// TIA Portal V16 export
// export: Created 2022-01-12T14:34:25.3404927Z, ExportSetting WithDefaults, DisplayName Totally Integrated Automation Portal, DisplayVersion V16 Update 4, DisplayName TIA Portal Version Control Interface, DisplayVersion V16 Update 2, DisplayName TIA Portal Openness, DisplayVersion V16 Update 4, DisplayName STEP 7 Professional, DisplayVersion V16 Update 4, DisplayName STEP 7 Safety, DisplayVersion V16, DisplayName WinCC Professional, DisplayVersion V16 Update 4
VAR_GLOBAL   // PLC tag table "Default tag table"
   System_Byte AT %MB1 : Byte;
   FirstScan AT %M1.0 : Bool;
   DiagStatusUpdate AT %M1.1 : Bool;
   AlwaysTRUE AT %M1.2 : Bool;
   AlwaysFALSE AT %M1.3 : Bool;
   Clock_Byte AT %MB0 : Byte;
   Clock_10Hz AT %M0.0 : Bool;
   Clock_5Hz AT %M0.1 : Bool;
   "Clock_2.5Hz" AT %M0.2 : Bool;
   Clock_2Hz AT %M0.3 : Bool;
   "Clock_1.25Hz" AT %M0.4 : Bool;
   Clock_1Hz AT %M0.5 : Bool;
   "Clock_0.625Hz" AT %M0.6 : Bool;
   "Clock_0.5Hz" AT %M0.7 : Bool;
   ala AT %MW2 : Int;
   "di24.2" AT %I0.2 : Bool;
   diSAFETY AT %I0.3 : Bool;
   diC201FC01 AT %I0.4 : Bool;
   diC202FC01 AT %I0.5 : Bool;
   diC202AV03c AT %I0.6 : Bool;
   diC202AV04c AT %I0.7 : Bool;
   diC201AV01c AT %I1.0 : Bool;
   diC201AV02c AT %I1.1 : Bool;
   diC202AV01c AT %I1.2 : Bool;
   diC202AV02c AT %I1.3 : Bool;
   diC211AV01c AT %I1.4 : Bool;
   diC212AV01c AT %I1.5 : Bool;
   diC2A1AV01c AT %I1.6 : Bool;
   diC2A1AV02c AT %I1.7 : Bool;
   diC2A1AV11c AT %I2.0 : Bool;
   diC2A1AV12c AT %I2.1 : Bool;
   diC2A1AV31c AT %I2.2 : Bool;
   diC2A1AV41c AT %I2.3 : Bool;
   diC2D1AV01c AT %I2.4 : Bool;
   diC2D1AV11c AT %I2.5 : Bool;
   diC2D1AV41c AT %I2.6 : Bool;
   diC2D1AV42c AT %I2.7 : Bool;
   diC2D2AV01c AT %I3.0 : Bool;
   diC2D2AV11c AT %I3.1 : Bool;
   diC2D2AV41c AT %I3.2 : Bool;
   diC2D2AV42c AT %I3.3 : Bool;
   diC2D3AV01c AT %I3.4 : Bool;
   diC2D3AV11c AT %I3.5 : Bool;
   diC2D3AV31c AT %I3.6 : Bool;
   diC2D3AV41c AT %I3.7 : Bool;
   diC2D3AV42c AT %I4.0 : Bool;
   diC2D3AV43c AT %I4.1 : Bool;
   diC2L1AV01c AT %I4.2 : Bool;
   diC2L1AV02c AT %I4.3 : Bool;
   diC2L1AV11c AT %I4.4 : Bool;
   diC2L1AV12c AT %I4.5 : Bool;
   diC2L1AV31c AT %I4.6 : Bool;
   diC2L1AV41c AT %I4.7 : Bool;
   diC2R1AV01c AT %I5.0 : Bool;
   diC2R1AV02c AT %I5.1 : Bool;
   diC2R1AV11c AT %I5.2 : Bool;
   diC2R1AV12c AT %I5.3 : Bool;
   diC2R1AV41c AT %I5.4 : Bool;
   diC2W1AV02c AT %I5.5 : Bool;
   diC2W1AV31c AT %I5.6 : Bool;
   diC2W1AV41c AT %I5.7 : Bool;
   diC211FV01 AT %I6.0 : Bool;
   diC212FV01 AT %I6.1 : Bool;
   diC2D1FV81 AT %I6.2 : Bool;
   diC2D2FV81 AT %I6.3 : Bool;
   diC2A1PD01 AT %I6.4 : Bool;
   diC2D1PD01 AT %I6.5 : Bool;
   diC2D2PD01 AT %I6.6 : Bool;
   diC2D3PD01 AT %I6.7 : Bool;
   diC2L1PD01 AT %I7.0 : Bool;
   diC2R1PD01 AT %I7.1 : Bool;
   diC2W1PD01 AT %I7.2 : Bool;
   diC2A1LL01 AT %I7.3 : Bool;
   diC2D1LL01 AT %I7.4 : Bool;
   diC2D2LL01 AT %I7.5 : Bool;
   diC2D3LL01 AT %I7.6 : Bool;
   diC2L1LL01 AT %I7.7 : Bool;
   diC2R1LL01 AT %I8.0 : Bool;
   diC2W1LL01 AT %I8.1 : Bool;
   diC2A1LH01 AT %I8.2 : Bool;
   diC2D1LH01 AT %I8.3 : Bool;
   diC2D2LH01 AT %I8.4 : Bool;
   diC2D3LH01 AT %I8.5 : Bool;
   diC2L1LH01 AT %I8.6 : Bool;
   diC2R1LH01 AT %I8.7 : Bool;
   diC2W1LH01 AT %I9.0 : Bool;
   doC201AV21b AT %Q0.0 : Bool;
   doC202AV21b AT %Q0.1 : Bool;
   doC2W1AV31b AT %Q0.2 : Bool;
   doC2W1AV02b AT %Q0.3 : Bool;
   doC2R1AV11b AT %Q0.4 : Bool;
   doC2R1AV12b AT %Q0.5 : Bool;
   doC2R1AV41b AT %Q0.6 : Bool;
   doC2R1AV01b AT %Q0.7 : Bool;
   doC2R1AV02b AT %Q1.0 : Bool;
   doC2L1AV11b AT %Q1.1 : Bool;
   doC2L1AV12b AT %Q1.2 : Bool;
   doC2L1AV41b AT %Q1.3 : Bool;
   doC2L1AV01b AT %Q1.4 : Bool;
   doC2L1AV02b AT %Q1.5 : Bool;
   doC2L1AV31b AT %Q1.6 : Bool;
   doC2A1AV11b AT %Q1.7 : Bool;
   doC2A1AV12b AT %Q2.0 : Bool;
   doC2A1AV41b AT %Q2.1 : Bool;
   doC2A1AV01b AT %Q2.2 : Bool;
   doC2A1AV02b AT %Q2.3 : Bool;
   doC2A1AV31b AT %Q2.4 : Bool;
   doC2D1AV11b AT %Q2.5 : Bool;
   doC2D1AV41b AT %Q2.6 : Bool;
   doC2D1AV42b AT %Q2.7 : Bool;
   doC2D1AV01b AT %Q3.0 : Bool;
   doC2D2AV01b AT %Q3.1 : Bool;
   doC2D2AV42b AT %Q3.2 : Bool;
   doC2D2AV41b AT %Q3.3 : Bool;
   doC2D2AV11b AT %Q3.4 : Bool;
   doC2D3AV41b AT %Q3.5 : Bool;
   doC2D3AV42b AT %Q3.6 : Bool;
   doC2D3AV11b AT %Q3.7 : Bool;
   doC2D3AV31b AT %Q4.0 : Bool;
   doC2D3AV43b AT %Q4.1 : Bool;
   doC2D3AV01b AT %Q4.2 : Bool;
   doC202AV01b AT %Q4.3 : Bool;
   doC202AV02b AT %Q4.4 : Bool;
   doC201AV01b AT %Q4.5 : Bool;
   doC201AV02b AT %Q4.6 : Bool;
   doC2A1AV42b AT %Q5.0 : Bool;
   doC2L1AV42b AT %Q5.1 : Bool;
   doC2D1AV81b AT %Q5.3 : Bool;
   doC2D2AV81b AT %Q5.4 : Bool;
   doC2W1AV41b AT %Q5.5 : Bool;
   doC211AV01b AT %Q5.6 : Bool;
   doC212AV01b AT %Q5.7 : Bool;
   doC202AV03b AT %Q6.0 : Bool;
   doC202AV04b AT %Q6.1 : Bool;
   doC2A1MP41b AT %Q6.6 : Bool;
   doC2L1MP41b AT %Q6.7 : Bool;
   doBuczek AT %Q7.0 : Bool;
   doZielona AT %Q7.1 : Bool;
   doCzerwona AT %Q7.2 : Bool;
   doZolta AT %Q7.3 : Bool;
   aiC2W1TT01 AT %IW10 : Int;
   aiC2R1TT01 AT %IW12 : Int;
   aiC2L1TT01 AT %IW14 : Int;
   aiC2A1TT01 AT %IW16 : Int;
   aiC2D1TT01 AT %IW18 : Int;
   aiC2D2TT01 AT %IW20 : Int;
   aiC2D3TT01 AT %IW22 : Int;
   aiC211TT01 AT %IW24 : Int;
   aiC212TT01 AT %IW26 : Int;
   aiC201TT01 AT %IW28 : Int;
   aiC202TT01 AT %IW30 : Int;
   aiC212QIC01 AT %IW32 : Int;
   aiC211QIC01 AT %IW34 : Int;
   aiC2A1LT01 AT %IW36 : Int;
   aiC2D1LT01 AT %IW38 : Int;
   aiC2D2LT01 AT %IW40 : Int;
   aiC2D3LT01 AT %IW42 : Int;
   aiC2L1LT01 AT %IW44 : Int;
   aiC2R1LT01 AT %IW46 : Int;
   aiC2W1LT01 AT %IW48 : Int;
   aoC201CV21 AT %QW8 : Int;
   aoC202CV21 AT %QW10 : Int;
   aoC201FC01 AT %QW12 : Int;
   aoC202FC01 AT %QW14 : Int;
   aoC2D1MP81 AT %QW16 : Int;
   aoC2D2MP81 AT %QW18 : Int;
   C202FT01volume AT %ID50 : Real;
   C201FT01volume AT %ID85 : Real;
   C202FT01temperature AT %ID120 : Real;
   C201FT01temperature AT %ID125 : Real;
   doC2A1AV43b AT %Q4.7 : Bool;
   doC2L1AV43b AT %Q5.2 : Bool;
   "di24.1" AT %I0.1 : Bool;
   C2L1MP41 AT %MW10 : Int;
   C2A1AV01 AT %MW94 : Int;
   C202AV01 AT %MW80 : Int;
   C2A1MP41 AT %MW8 : Int;
   C2A1AV41 AT %MW104 : Int;
   C2D1FV81 AT %MW70 : Int;
   C2W1LL01 AT %MW62 : Int;
   C2D1PD01 AT %MW30 : Int;
   C2R1LL01 AT %MW56 : Int;
   C2D3PD01 AT %MW44 : Int;
   C2D3LL01 AT %MW42 : Int;
   C2L1AV43 AT %MW110 : Int;
   C201AV21 AT %MW78 : Int;
   C2A1PD01 AT %MW22 : Int;
   C2W1PD01 AT %MW64 : Int;
   C2D2FV81 AT %MW72 : Int;
   C202AV02 AT %MW82 : Int;
   C211AV01 AT %MW90 : Int;
   C2L1LH01 AT %MW46 : Int;
   C2D2LH01 AT %MW32 : Int;
   C2D1AV01 AT %MW112 : Int;
   diC2D2LL81 AT %I9.4 : Bool;
   C202AV21 AT %MW88 : Int;
   C2L1Ll41 AT %MW50 : Int;
   C212AV01 AT %MW92 : Int;
   C2A1AV12 AT %MW100 : Int;
   C211FV01 AT %MW66 : Int;
   C2R1PD01 AT %MW58 : Int;
   C2A1AV42 AT %MW106 : Int;
   diC2D1LL81 AT %I9.3 : Bool;
   C202FC01 AT %MW4 : Int;
   C2L1Ll01 AT %MW48 : Int;
   diC2A1LL41 AT %I9.1 : Bool;
   diC2L1LL41 AT %I9.2 : Bool;
   C2A1LH01 AT %MW16 : Int;
   C202AV03 AT %MW84 : Int;
   C2D2MP81 AT %MW14 : Int;
   C2D2LL01 AT %MW34 : Int;
   C2L1PD01 AT %MW52 : Int;
   C2D1LL81 AT %MW28 : Int;
   C2W1LH01 AT %MW60 : Int;
   C2A1AV02 AT %MW96 : Int;
   C2R1LH01 AT %MW54 : Int;
   C201AV01 AT %MW74 : Int;
   C2D1LH01 AT %MW24 : Int;
   C2D1LL01 AT %MW26 : Int;
   C2A1LL41 AT %MW20 : Int;
   C202AV04 AT %MW86 : Int;
   C212FV01 AT %MW68 : Int;
   C2D1MP81 AT %MW12 : Int;
   C2A1LL01 AT %MW18 : Int;
   C2A1AV31 AT %MW102 : Int;
   C2D2PD01 AT %MW38 : Int;
   C201AV02 AT %MW76 : Int;
   C2D3LH01 AT %MW40 : Int;
   C2D2LL81 AT %MW36 : Int;
   C2A1AV11 AT %MW98 : Int;
   C2A1AV43 AT %MW108 : Int;
   C2D1AV41 AT %MW116 : Int;
   C2L1AV31 AT %MW152 : Int;
   C2L1AV41 AT %MW154 : Int;
   C2R1AV12 AT %MW164 : Int;
   C211QIC01 AT %MW218 : Int;
   CD1LT01 AT %MW198 : Int;
   C2D3AV11 AT %MW134 : Int;
   C2L1AV01 AT %MW144 : Int;
   C2L1AV12 AT %MW150 : Int;
   C2L1AV11 AT %MW148 : Int;
   C2D3TT01 AT %MW186 : Int;
   CD2LT01 AT %MW200 : Int;
   C2D1AV81 AT %MW120 : Int;
   C2D1TT01 AT %MW182 : Int;
   C201CV21 AT %MW220 : Int;
   C2L1LT01 AT %MW210 : Int;
   C2D3AV42 AT %MW140 : Int;
   C211TT01 AT %MW188 : Int;
   C2D2AV41 AT %MW126 : Int;
   C2D2AV01 AT %MW122 : Int;
   C2D2LT01 AT %MW204 : Int;
   C2D3AV01 AT %MW132 : Int;
   C2W1LT01 AT %MW214 : Int;
   CD3LT01 AT %MW202 : Int;
   C2D2AV42 AT %MW128 : Int;
   C2R1LT01 AT %MW212 : Int;
   C2D2TT01 AT %MW184 : Int;
   C2A1LT01 AT %MW196 : Int;
   C202TT01 AT %MW194 : Int;
   C2L1TT01 AT %MW178 : Int;
   C2R1AV01 AT %MW158 : Int;
   C2D1LT01 AT %MW208 : Int;
   C212TT01 AT %MW190 : Int;
   C212QIC01 AT %MW216 : Int;
   C2D2AV11 AT %MW124 : Int;
   C201TT01 AT %MW192 : Int;
   C2D3AV31 AT %MW136 : Int;
   C2D3LT01 AT %MW206 : Int;
   C2RW1AV31 AT %MW170 : Int;
   C2A1TT01 AT %MW180 : Int;
   C202CV21 AT %MW222 : Int;
   C2R1AV11 AT %MW162 : Int;
   C2RW1AV02 AT %MW168 : Int;
   C2D3AV41 AT %MW138 : Int;
   C2L1AV02 AT %MW146 : Int;
   C2R1TT01 AT %MW176 : Int;
   C2R1AV41 AT %MW166 : Int;
   C2RW1AV41 AT %MW172 : Int;
   C2D1AV42 AT %MW118 : Int;
   C2W1TT01 AT %MW174 : Int;
   C2R1AV02 AT %MW160 : Int;
   C2D2AV81 AT %MW130 : Int;
   C2D3AV43 AT %MW142 : Int;
   C2D1AV11 AT %MW114 : Int;
   C2L1AV42 AT %MW156 : Int;
   staryNumerObiektuWybranyZHMI AT %MW226 : Int;
   numerObiektuWybranyZHMI AT %MW224 : Int;
   doC2W1AV01b AT %Q7.4 : Bool;
   C2W1AV01 AT %MW228 : Int;
   diC2W1AV01c AT %I9.7 : Bool;
   C2W1AV02 AT %MW230 : Int;
   doC2D2MP81 AT %Q6.3 : Bool;
   doC202FC01 AT %Q6.5 : Bool;
   doC2D1MP81 AT %Q6.2 : Bool;
   doC201FC01 AT %Q6.4 : Bool;
   hmi_alarm AT %M232.0 : Bool;
   C2W1AV41 AT %MW236 : Int;
   C2W1AV31 AT %MW234 : Int;
   "Cip1.pompaPodawaniaCip" AT %MW6 : Int;
   linia1_pompa_zezwolenie AT %M232.1 : Bool;
   krokZapauzowany AT %MW238 : Int;
   numer_kroku_stary_1 AT %MW240 : Int;
   numer_kroku_stary_2 AT %MW242 : Int;
END_VAR
VAR_GLOBAL CONSTANT   // user constants
   f101fc01 : Int := 2;
END_VAR
